// TIA Portal V17 export
// export: Created 2022-05-02T08:04:29.8806059Z, ExportSetting WithDefaults, DisplayName Totally Integrated Automation Portal, DisplayVersion V17 Update 3, DisplayName TIA Portal Openness, DisplayVersion V17 Update 3, DisplayName TIA Portal Teamcenter Gateway, DisplayVersion V17 Update 3, DisplayName TIA Portal Version Control Interface, DisplayVersion V17, DisplayName SINAMICS Startdrive Advanced, DisplayVersion V17 Update2, DisplayName SINAMICS Startdrive G130, G150, S120, S150, SINAMICS MV, S210, DisplayVersion V17 Update2, DisplayName SINAMICS Startdrive G110M, G120, G120C, G120D, G120P, G115D, DisplayVersion V17 Update2, DisplayName STEP 7 Professional, DisplayVersion V17 Update 3, DisplayName STEP 7 CFC, DisplayVersion V17 Update 1, DisplayName STEP 7 Safety, DisplayVersion V17, DisplayName WinCC UA Professional, DisplayVersion V17 Update 3, DisplayName WinCC Unified Calendar, DisplayVersion V17, DisplayName WinCC Unified Performance Insight, DisplayVersion V17
DATA_BLOCK "DB_CALCUL"   // DB37
{ S7_Optimized_Access := 'TRUE' }
VERSION : 0.1
// stored: AutoNumber true, DBAccessibleFromOPCUA true, DBAccessibleFromWebserver true, IsOnlyStoredInLoadMemory false, IsRetainMemResEnabled false, IsWriteProtectedInAS false, MemoryReserve 0
   VAR
      DATA_Int1 : Int := 0;
      DATA_Int2 : Int;
      DATA_Int3 : Int;
      DATA_Real : Real;
      DATA_Result : Real;
   END_VAR
BEGIN
END_DATA_BLOCK
